(*
SPDX-FileCopyrightText: © 2026 Oleksandr Tiutyk <trofimich@gmail.com>
SPDX-License-Identifier: MIT
License: https://opensource.org/license/mit
*)

(*!
<summary>Reports that destination storage cannot hold the requested result.</summary>
<description>
The caller detects the condition; this exception does not inspect or modify the collection or destination.
Uses the GeneralException task-local cycle lifetime and throw rules. Dynamic copies are explicitly registered
by Clone after construction; plain __NEW does not transfer ownership to the task manager.
</description>
*)

{attribute 'enable_dynamic_creation'}
{attribute 'no_explicit_call' := 'do not call this function block directly'}
FUNCTION_BLOCK TargetVariableMemoryOverflowException EXTENDS GeneralException IMPLEMENTS ITargetVariableMemoryOverflowException
VAR_STAT
	//! <summary>Class name shared by all instances of this function block.</summary>
	{attribute 'hide'} 
	_ClassName : STRING := __POUNAME();
END_VAR

{attribute 'monitoring' := 'call'}
PROPERTY ClassName : REFERENCE TO STRING
GET
ClassName REF= _ClassName;
END_GET
END_PROPERTY

(*!
<summary>Creates a clone of this concrete exception type.</summary>
<description>
Copies GeneralException fields and timestamps. The clone belongs to DynamicMemoryManager until cleanup of the
creating task; callers must not delete it. Allocation failure is terminal. Registers the newly constructed
instance before copying payload, outside FB_init. Registration failure releases the unregistered instance and
raises a terminal error; copy failure leaves the registered instance owned by the task manager for cleanup.
Custom overrides must follow the same ownership sequence.
</description>
*)
METHOD Clone : IObject
VAR
	exceptionClone : POINTER TO TargetVariableMemoryOverflowException;
END_VAR
exceptionClone := __NEW(TargetVariableMemoryOverflowException);

IF exceptionClone = 0 THEN
	DynamicMemoryManager.RaiseAllocationFailure();
END_IF

DynamicMemoryManager.RegisterAutoDisposedObject(autoDisposedObject := exceptionClone^);

exceptionClone^.CopyGeneralFields(sourceException := THIS^);

Clone := exceptionClone^;
END_METHOD

(*!
<summary>Provides the library namespace used in diagnostics.</summary>
<description>
Borrowed read-only reference to the compiler-initialized library namespace; no ownership transfer.
</description>
*)
{attribute 'monitoring' := 'call'}
PROPERTY NamespaceName : REFERENCE TO STRING
GET
NamespaceName REF= CurrentNamespace.Name;
END_GET
END_PROPERTY

(*!
<summary>Reports the byte size of this concrete instance.</summary>
<description>
Uses XSIZEOF on the instance. Does not include separately allocated payloads or prove that an arbitrary
address is valid.
</description>
*)
{attribute 'monitoring' := 'call'}
PROPERTY SelfSize : ULINT
GET
SelfSize := XSIZEOF(THIS^);
END_GET
END_PROPERTY

(*!
<summary>Builds the diagnostic and raises this exception through GeneralException.</summary>
<description>
Copies the supplied diagnostic data without heap allocation during message preparation, sets error code to
zero and supplies no inner exception. Call only in a cyclic task, not during FB_init. The caller must already
have detected the reported condition.
</description>
<param name="targetVariableName">Destination name used in the diagnostic.</param>
<param name="targetVariableSize">
Available destination storage in bytes, including string terminator storage where applicable.
</param>
*)
METHOD Throw
VAR_INPUT
	sourceNamespaceName : STRING;
	sourceClassName : STRING;
	sourcePOUName : STRING;
	sourcePosition : STRING;
	targetVariableName : STRING;
	targetVariableSize : ULINT;
END_VAR
VAR
	message : ERROR_MESSAGE;
END_VAR
WideStrings.Append255(
	message,
	"Terget variable '",
	TO_WSTRING(targetVariableName),
	"' (size ",
	TO_WSTRING(targetVariableSize),
	") memory overflow '",
	TO_WSTRING(GetFullPOUName(
		sourceNamespaceName := sourceNamespaceName,
		sourceClassName := sourceClassName,
		sourcePOUName := sourcePOUName
	)),
	"'");

InternalThrow(
	sourceNamespaceName := sourceNamespaceName,
	sourceClassName := sourceClassName,
	sourcePOUName := sourcePOUName,
	sourcePosition := sourcePosition,
	message := message,
	errorCode := 0,
	innerException := 0
);
END_METHOD

END_FUNCTION_BLOCK

(* stored: Version 1.1.0.1
   POU TargetVariableMemoryOverflowException: Id {a5c51537-9964-43b1-bc8c-6a2ce7304192}, SpecialFunc None
   Property ClassName: Id {6face4de-0106-4653-8501-0739f37c18e9}
   Get Get: Id {30d770a2-ebf9-4246-aef6-3271c58673ee}
   Method Clone: Id {9ed41139-91ec-41da-8fa6-2f309f22fbed}
   Property NamespaceName: Id {8f8de7c2-c18d-4fe8-b545-c99ae3e41e03}
   Get Get: Id {f1c191f8-a27e-4544-9f9e-1a0a2920d846}
   Property SelfSize: Id {2752ec58-dcee-4d7a-8f6b-d4e2f3b6d8fd}
   Get Get: Id {e13fa4a6-88b7-4506-b77e-187869e9727d}
   Method Throw: Id {c8177a3a-3507-4fd9-82e5-01f82a5acc18} *)
